// TIA Portal V17 export
// export: Created 2025-07-01T09:58:31.7616541Z, ExportSetting WithDefaults, DisplayName Totally Integrated Automation Portal, DisplayVersion V17 Update 8, DisplayName TIA Portal Openness, DisplayVersion V17 Update 8, DisplayName TIA Portal Version Control Interface, DisplayVersion V17, DisplayName SINAMICS Startdrive Advanced, DisplayVersion V17 SP2, DisplayName SINAMICS Startdrive G110M, G120, G120C, G120D, G120P, G115D, DisplayVersion V17 SP2, DisplayName SINAMICS Startdrive G130, G150, S120, S150, SINAMICS MV, S210, DisplayVersion V17 SP2, DisplayName STEP 7 Professional, DisplayVersion V17 Update 8, DisplayName SINUMERIK ONE STEP 7 Toolbox, DisplayVersion V17 Update 12, DisplayName SINUMERIK ONE PLC Basic Program Plus, DisplayVersion V17 Update 12, DisplayName SINUMERIK 840D sl STEP 7 Toolbox, DisplayVersion V17 Update 12, DisplayName STEP 7 Safety, DisplayVersion V17 Update 6, DisplayName WinCC Advanced, DisplayVersion V17 Update 8
FUNCTION "FC301_ALARMS_OPERATOR_HELP" : Void   // FC301, LAD
{ S7_Optimized_Access := 'TRUE' }
VERSION : 0.1
// stored: AutoNumber false, IsIECCheckEnabled false, SetENOAutomatically false, UDAEnableTagReadback false
   VAR_TEMP
      PART_TYPE : Int;
   END_VAR
   VAR_TEMP   // added for the SCL form of the ladder/FBD networks
      _w1 : Bool;
   END_VAR
BEGIN

REGION Network 1: FC421 HOLA PC ALARM
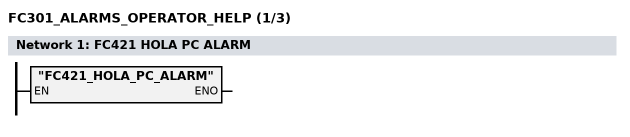
   RUNG wire#powerrail
      "FC421_HOLA_PC_ALARM"()
   END_RUNG
   // the same network as SCL:
   "FC421_HOLA_PC_ALARM"();
END_REGION

REGION Network 2: OPERATOR HELP
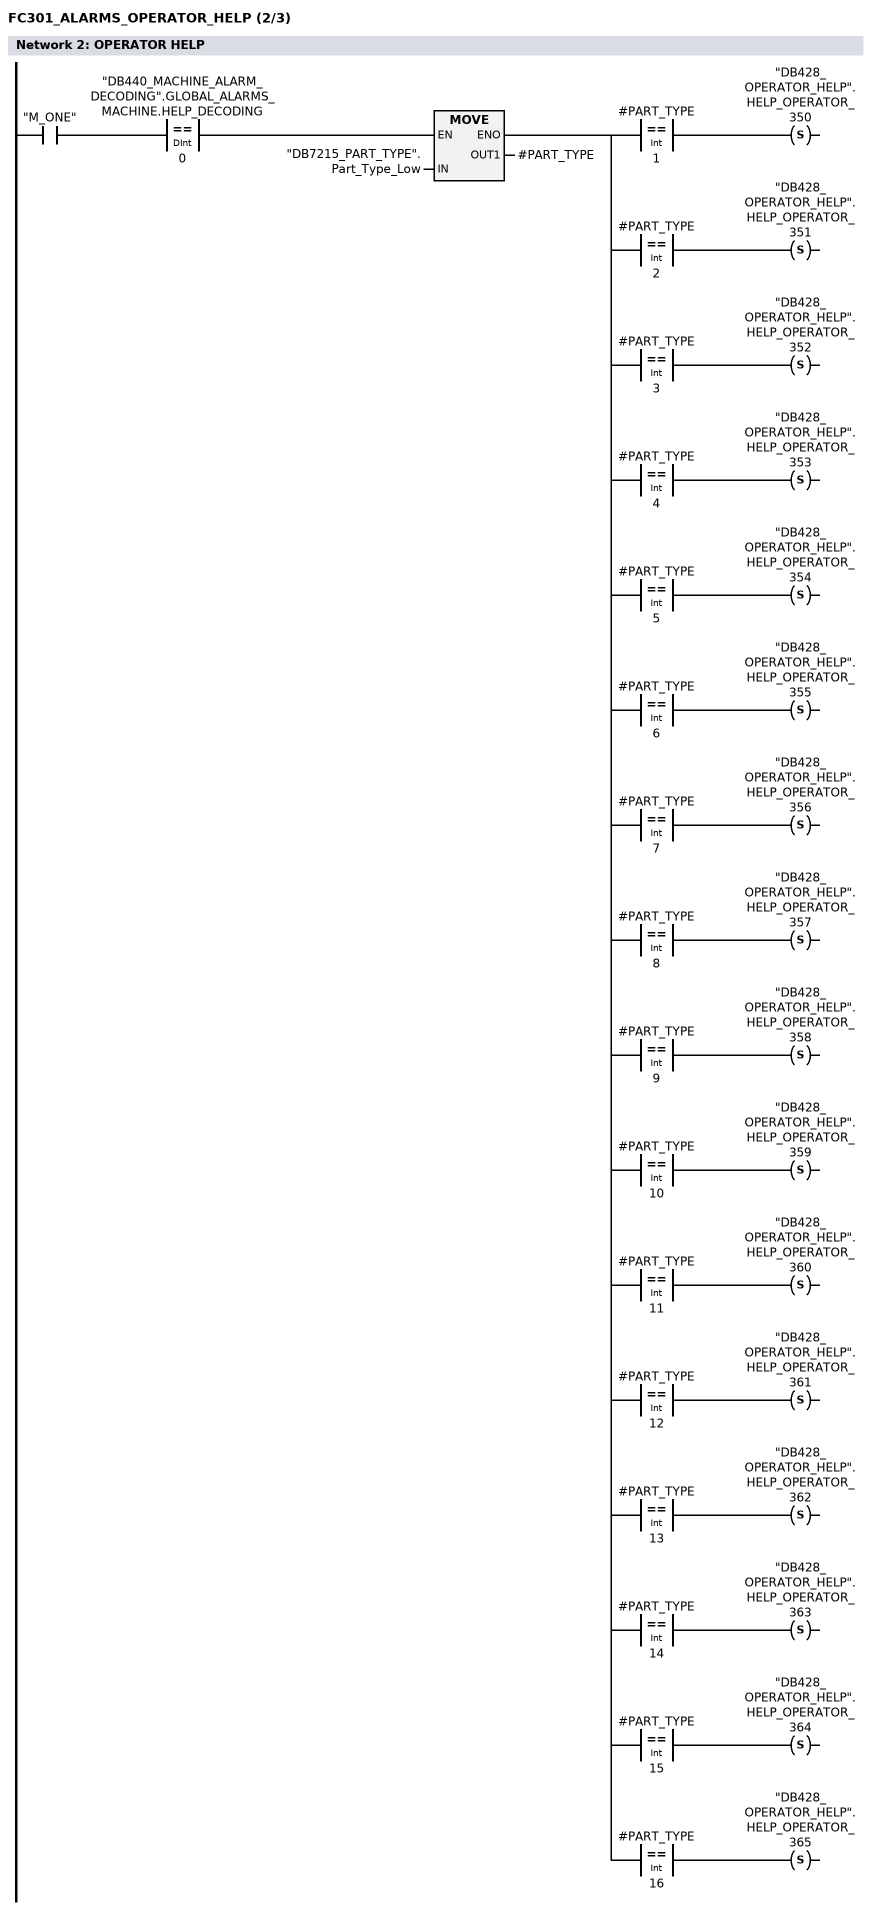
   RUNG wire#powerrail
      Contact( "M_ONE" )
      { S7_Templates := "SrcType := DInt" } EQ_Contact(in1 := "DB440_MACHINE_ALARM_DECODING".GLOBAL_ALARMS_MACHINE.HELP_DECODING, in2 := 0)
      { S7_GenerateENO := "TRUE" } Move(in := "DB7215_PART_TYPE".Part_Type_Low, out1 => #PART_TYPE)
      wire#w1
      { S7_Templates := "SrcType := Int" } EQ_Contact(in1 := #PART_TYPE, in2 := 1)
      S_Coil( "DB428_OPERATOR_HELP".HELP_OPERATOR_350 )
   END_RUNG
   RUNG wire#w1
      { S7_Templates := "SrcType := Int" } EQ_Contact(in1 := #PART_TYPE, in2 := 2)
      S_Coil( "DB428_OPERATOR_HELP".HELP_OPERATOR_351 )
   END_RUNG
   RUNG wire#w1
      { S7_Templates := "SrcType := Int" } EQ_Contact(in1 := #PART_TYPE, in2 := 3)
      S_Coil( "DB428_OPERATOR_HELP".HELP_OPERATOR_352 )
   END_RUNG
   RUNG wire#w1
      { S7_Templates := "SrcType := Int" } EQ_Contact(in1 := #PART_TYPE, in2 := 4)
      S_Coil( "DB428_OPERATOR_HELP".HELP_OPERATOR_353 )
   END_RUNG
   RUNG wire#w1
      { S7_Templates := "SrcType := Int" } EQ_Contact(in1 := #PART_TYPE, in2 := 5)
      S_Coil( "DB428_OPERATOR_HELP".HELP_OPERATOR_354 )
   END_RUNG
   RUNG wire#w1
      { S7_Templates := "SrcType := Int" } EQ_Contact(in1 := #PART_TYPE, in2 := 6)
      S_Coil( "DB428_OPERATOR_HELP".HELP_OPERATOR_355 )
   END_RUNG
   RUNG wire#w1
      { S7_Templates := "SrcType := Int" } EQ_Contact(in1 := #PART_TYPE, in2 := 7)
      S_Coil( "DB428_OPERATOR_HELP".HELP_OPERATOR_356 )
   END_RUNG
   RUNG wire#w1
      { S7_Templates := "SrcType := Int" } EQ_Contact(in1 := #PART_TYPE, in2 := 8)
      S_Coil( "DB428_OPERATOR_HELP".HELP_OPERATOR_357 )
   END_RUNG
   RUNG wire#w1
      { S7_Templates := "SrcType := Int" } EQ_Contact(in1 := #PART_TYPE, in2 := 9)
      S_Coil( "DB428_OPERATOR_HELP".HELP_OPERATOR_358 )
   END_RUNG
   RUNG wire#w1
      { S7_Templates := "SrcType := Int" } EQ_Contact(in1 := #PART_TYPE, in2 := 10)
      S_Coil( "DB428_OPERATOR_HELP".HELP_OPERATOR_359 )
   END_RUNG
   RUNG wire#w1
      { S7_Templates := "SrcType := Int" } EQ_Contact(in1 := #PART_TYPE, in2 := 11)
      S_Coil( "DB428_OPERATOR_HELP".HELP_OPERATOR_360 )
   END_RUNG
   RUNG wire#w1
      { S7_Templates := "SrcType := Int" } EQ_Contact(in1 := #PART_TYPE, in2 := 12)
      S_Coil( "DB428_OPERATOR_HELP".HELP_OPERATOR_361 )
   END_RUNG
   RUNG wire#w1
      { S7_Templates := "SrcType := Int" } EQ_Contact(in1 := #PART_TYPE, in2 := 13)
      S_Coil( "DB428_OPERATOR_HELP".HELP_OPERATOR_362 )
   END_RUNG
   RUNG wire#w1
      { S7_Templates := "SrcType := Int" } EQ_Contact(in1 := #PART_TYPE, in2 := 14)
      S_Coil( "DB428_OPERATOR_HELP".HELP_OPERATOR_363 )
   END_RUNG
   RUNG wire#w1
      { S7_Templates := "SrcType := Int" } EQ_Contact(in1 := #PART_TYPE, in2 := 15)
      S_Coil( "DB428_OPERATOR_HELP".HELP_OPERATOR_364 )
   END_RUNG
   RUNG wire#w1
      { S7_Templates := "SrcType := Int" } EQ_Contact(in1 := #PART_TYPE, in2 := 16)
      S_Coil( "DB428_OPERATOR_HELP".HELP_OPERATOR_365 )
   END_RUNG
   // the same network as SCL:
   // ENO of a box is taken as its EN; it also drops when the box reports an error
   #_w1 := "M_ONE" AND ("DB440_MACHINE_ALARM_DECODING".GLOBAL_ALARMS_MACHINE.HELP_DECODING = 0);
   IF #_w1 THEN #PART_TYPE := "DB7215_PART_TYPE".Part_Type_Low; END_IF;
   IF #_w1 AND (#PART_TYPE = 1) THEN "DB428_OPERATOR_HELP".HELP_OPERATOR_350 := TRUE; END_IF;
   IF #_w1 AND (#PART_TYPE = 2) THEN "DB428_OPERATOR_HELP".HELP_OPERATOR_351 := TRUE; END_IF;
   IF #_w1 AND (#PART_TYPE = 3) THEN "DB428_OPERATOR_HELP".HELP_OPERATOR_352 := TRUE; END_IF;
   IF #_w1 AND (#PART_TYPE = 4) THEN "DB428_OPERATOR_HELP".HELP_OPERATOR_353 := TRUE; END_IF;
   IF #_w1 AND (#PART_TYPE = 5) THEN "DB428_OPERATOR_HELP".HELP_OPERATOR_354 := TRUE; END_IF;
   IF #_w1 AND (#PART_TYPE = 6) THEN "DB428_OPERATOR_HELP".HELP_OPERATOR_355 := TRUE; END_IF;
   IF #_w1 AND (#PART_TYPE = 7) THEN "DB428_OPERATOR_HELP".HELP_OPERATOR_356 := TRUE; END_IF;
   IF #_w1 AND (#PART_TYPE = 8) THEN "DB428_OPERATOR_HELP".HELP_OPERATOR_357 := TRUE; END_IF;
   IF #_w1 AND (#PART_TYPE = 9) THEN "DB428_OPERATOR_HELP".HELP_OPERATOR_358 := TRUE; END_IF;
   IF #_w1 AND (#PART_TYPE = 10) THEN "DB428_OPERATOR_HELP".HELP_OPERATOR_359 := TRUE; END_IF;
   IF #_w1 AND (#PART_TYPE = 11) THEN "DB428_OPERATOR_HELP".HELP_OPERATOR_360 := TRUE; END_IF;
   IF #_w1 AND (#PART_TYPE = 12) THEN "DB428_OPERATOR_HELP".HELP_OPERATOR_361 := TRUE; END_IF;
   IF #_w1 AND (#PART_TYPE = 13) THEN "DB428_OPERATOR_HELP".HELP_OPERATOR_362 := TRUE; END_IF;
   IF #_w1 AND (#PART_TYPE = 14) THEN "DB428_OPERATOR_HELP".HELP_OPERATOR_363 := TRUE; END_IF;
   IF #_w1 AND (#PART_TYPE = 15) THEN "DB428_OPERATOR_HELP".HELP_OPERATOR_364 := TRUE; END_IF;
   IF #_w1 AND (#PART_TYPE = 16) THEN "DB428_OPERATOR_HELP".HELP_OPERATOR_365 := TRUE; END_IF;
END_REGION

REGION Network 3: CALL FC428 OPERATOR HELP
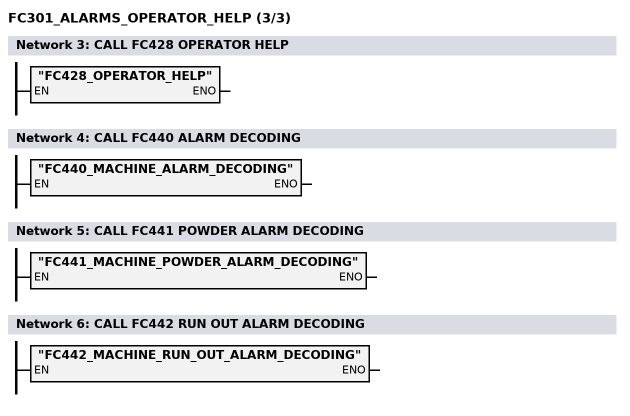
   RUNG wire#powerrail
      "FC428_OPERATOR_HELP"()
   END_RUNG
   // the same network as SCL:
   "FC428_OPERATOR_HELP"();
END_REGION

REGION Network 4: CALL FC440 ALARM DECODING
   RUNG wire#powerrail
      "FC440_MACHINE_ALARM_DECODING"()
   END_RUNG
   // the same network as SCL:
   "FC440_MACHINE_ALARM_DECODING"();
END_REGION

REGION Network 5: CALL FC441 POWDER ALARM DECODING
   RUNG wire#powerrail
      "FC441_MACHINE_POWDER_ALARM_DECODING"()
   END_RUNG
   // the same network as SCL:
   "FC441_MACHINE_POWDER_ALARM_DECODING"();
END_REGION

REGION Network 6: CALL FC442 RUN OUT ALARM DECODING
   RUNG wire#powerrail
      "FC442_MACHINE_RUN_OUT_ALARM_DECODING"()
   END_RUNG
   // the same network as SCL:
   "FC442_MACHINE_RUN_OUT_ALARM_DECODING"();
END_REGION
END_FUNCTION
